PROGRAM MAIN
VAR
END_VAR

opcua.bBool1 := opcua.bBool2;
opcua.iInt3 := opcua.iInt1 + opcua.iInt2;

END_PROGRAM

(* stored: Version 1.1.0.1, ProductVersion 3.1.4024.10
   POU MAIN: Id {fbe3430b-38fb-48c9-bd12-bf601457e4f2}, SpecialFunc None *)
